FUNCTION_BLOCK SS5a_Ejector (* Basic FB with empty ECC *)
  (* Standard: 61499-2 *)
  (* Version 1.0, 2024-10-03, DEVIASH *)
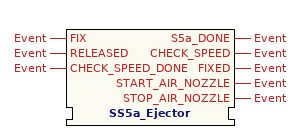
  EVENT_INPUT
    FIX;
    RELEASED;
    CHECK_SPEED_DONE;
  END_EVENT
  EVENT_OUTPUT
    S5a_DONE;
    CHECK_SPEED;
    FIXED;
    START_AIR_NOZZLE;
    STOP_AIR_NOZZLE;
  END_EVENT
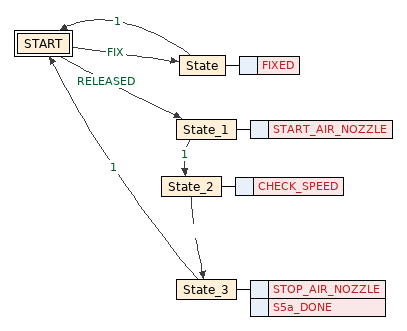
  EC_STATES
    START; (* Initial State *)
    State : -> FIXED;
    State_1 : -> START_AIR_NOZZLE;
    State_2 : -> CHECK_SPEED;
    State_3 : -> STOP_AIR_NOZZLE, -> S5a_DONE;
  END_STATES
  EC_TRANSITIONS
    START TO State := FIX;
    State TO START := 1;
    START TO State_1 := RELEASED;
    State_1 TO State_2 := 1;
    State_2 TO State_3 := ;
    State_3 TO START := 1;
  END_TRANSITIONS
END_FUNCTION_BLOCK
